FUNCTION_BLOCK FB_StateMachine // A basic statemachine with some convenient outputs
VAR CONSTANT
	MAX_TIME : TIME := UDINT_TO_TIME(16#FFFFFFFF);
END_VAR
VAR_IN_OUT
	nState : UDINT;
END_VAR
VAR_OUTPUT
	tTimeInState : TIME;
	bStateChanged : BOOL;
END_VAR
VAR
	nStatePrev : UDINT;
	tonTimeInState : TON;
END_VAR

bStateChanged := (nStatePrev <> nState);
nStatePrev := nState;
tonTimeInState(IN := NOT bStateChanged, PT := MAX_TIME);
tTimeInState := tonTimeInState.ET;

END_FUNCTION_BLOCK

(* stored: Version 1.1.0.1, ProductVersion 3.1.4024.11
   POU FB_StateMachine: Id {b37487b3-c0ea-0602-0c95-36b38859673c}, SpecialFunc None *)
